// TIA Portal V17 export
// export: Created 2023-02-25T16:31:53.2453939Z, ExportSetting WithDefaults, DisplayName Totally Integrated Automation Portal, DisplayVersion V17, DisplayName TIA Portal Openness, DisplayVersion V17, DisplayName TIA Portal Version Control Interface, DisplayVersion V17, DisplayName TIA Portal Test Suite Advanced, DisplayVersion V17, DisplayName STEP 7 Professional, DisplayVersion V17, DisplayName SIMATIC Energy Suite, DisplayVersion V17, DisplayName STEP 7 Safety, DisplayVersion V17, DisplayName WinCC Professional, DisplayVersion V17
FUNCTION "LOG_ButtonsLight" : Void   // FC14, LAD
{ S7_Optimized_Access := 'TRUE' }
VERSION : 0.1
// stored: AutoNumber true, IsIECCheckEnabled false, SetENOAutomatically false, UDAEnableTagReadback false
BEGIN

REGION Network 1: Button Start
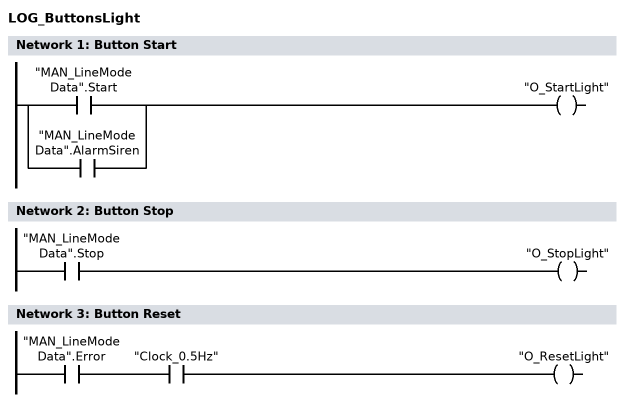
   RUNG wire#powerrail
      Contact( "MAN_LineModeData".Start )
      wire#w1
      Coil( "O_StartLight" )
   END_RUNG
   RUNG wire#powerrail
      Contact( "MAN_LineModeData".AlarmSiren )
   END_RUNG wire#w1
   // the same network as SCL:
   "O_StartLight" := "MAN_LineModeData".Start OR "MAN_LineModeData".AlarmSiren;
END_REGION

REGION Network 2: Button Stop
   RUNG wire#powerrail
      Contact( "MAN_LineModeData".Stop )
      Coil( "O_StopLight" )
   END_RUNG
   // the same network as SCL:
   "O_StopLight" := "MAN_LineModeData".Stop;
END_REGION

REGION Network 3: Button Reset
   RUNG wire#powerrail
      Contact( "MAN_LineModeData".Error )
      Contact( "Clock_0.5Hz" )
      Coil( "O_ResetLight" )
   END_RUNG
   // the same network as SCL:
   "O_ResetLight" := "MAN_LineModeData".Error AND "Clock_0.5Hz";
END_REGION
END_FUNCTION
